// TIA Portal V20 export
VAR_GLOBAL   // PLC tag table "cmd"
END_VAR
VAR_GLOBAL CONSTANT   // user constants
   cmd_acquired : Int := 1;
   cmd_executing : Int := 2;
   cmd_executed : Int := 3;
   cmd_aborted : Int := 4;
   cmd_rejected : Int := 5;
   cmd_waitingNewCmd : Int := 0;
END_VAR
